// TwinCAT 3 PLC project Tc3_Logging
// Title: Tc3_Logging
// Company: www.peterzerlauth.com
// Author: Peter Zerlauth
// ProjectVersion: 0.0.0.8
// Description: Tc3_Logging – TwinCAT 3 Event Logging Framework Copyright (c) Peter Zerlauth This component is provided under a Dual Licensing Model: 1. GPLv3 Open-Source License - Free for personal, educational, and non-commercial use. - Commercial use allowed only if the entire application is published under GPLv3, including all modifications to this code. - Requires full disclosure of source code for derivative works. 2. Commercial License - Required for integration into proprietary or closed-source products. - Removes all GPLv3 copyleft obligations. - Includes optional warranty, professional support, and long-term maintenance options. For commercial licensing, contact: info@peterzerlauth.com By using this Function Block you agree to the terms of the selected license.
// ProgramVersion: 3.1.4026.24
// libraries:
//   SysDir, * (System)
//   SysFile, * (System)
//   Tc2_Standard, * (Beckhoff Automation GmbH)
//   Tc2_System, * (Beckhoff Automation GmbH)
//   Tc2_Utilities, * (Beckhoff Automation GmbH)
//   Tc3_EventLogger, * (Beckhoff Automation GmbH)
//   Tc3_Module, * (Beckhoff Automation GmbH)
// project tree:
//   Argument/ FB_Argument.TcPOU, I_Argument.TcIO
//   Event/ I_Event.TcIO (not stored), FB_Event.TcPOU (not stored)
//   Global Variables/ GVL.TcGVL
//   Helpers/File/ E_FileState.TcDUT, FB_File.TcPOU, I_File.TcIO
//   Helpers/ F_Filter.TcPOU, F_Hash.TcPOU, F_InstancePath.TcPOU, F_Log.TcPOU, F_Print.TcPOU, F_Remove.TcPOU, LogLevel_To_Severity.TcPOU
//   Logger/ E_LogLevel.TcDUT, I_Logger.TcIO
//   Logger/FileLogger/ FB_FileLogger.TcPOU
//   Logger/HmiLogger/ FB_HmiLogger.TcPOU
//   Logger/Manager/ FB_LoggerManager.TcPOU
//   Logger/TcLogger/ FB_TcLogger.TcPOU
//   Message/ FB_Message.TcPOU
//   Project Information/ F_GetCompany.TcPOU, F_GetTitle.TcPOU, F_GetVersion.TcPOU
//   Version/ Global_Version.TcGVL
// (motion and I/O tree: see PLC project plc01)
// real-time tasks:
//   TASK SlowTask: cycle T#20ms, priority 20, ADS port 350
//   TASK FastTask: cycle T#1ms, priority 1, ADS port 351

// ---- Helpers/File/E_FileState.TcDUT
{attribute 'qualified_only'}
{attribute 'strict'}
{attribute 'to_string'}
TYPE E_FileState :
(
    OK := 0,             // File could be opened
    NO_FILE := 1,        // No file available
    ILLEGAL_POS := 2,    // Illegal position in the file
    FULL := 3,           // No more space on the filesystem
    EOF := 4             // End of file reached
) UDINT;
END_TYPE

// ---- Logger/E_LogLevel.TcDUT
{attribute 'qualified_only'}
{attribute 'strict'}
{attribute 'to_string'}
TYPE E_LogLevel :
(
    Verbose 	:= 1,
    Info  		:= 2,
    Warning  	:= 3,
    Error 		:= 4,
    Critical 	:= 5
);
END_TYPE

// ---- Global Variables/GVL.TcGVL
{attribute 'no-analysis'}
{attribute 'qualified_only'} 
VAR_GLOBAL
	{attribute 'hide'} 
	aBuffer:				ARRAY[0..99] OF FB_Message;
	{attribute 'hide'} 
    nBuffer:				UINT := 0;
	{attribute 'hide'} 
	nTimestamp:				Tc2_Utilities.T_FILETIME64;	
	{attribute 'hide'} 
	nFunction:				Tc2_Utilities.T_FILETIME64;		
END_VAR

// ---- Version/Global_Version.TcGVL
{attribute 'TcGenerated'}
{attribute 'no-analysis'}
{attribute 'linkalways'}
// This function has been automatically generated from the project information.
VAR_GLOBAL CONSTANT
	{attribute 'const_non_replaced'}
	stLibVersion_Tc3_Logging : ST_LibVersion := (iMajor := 0, iMinor := 0, iBuild := 0, iRevision := 8, nFlags := 0, sVersion := '0.0.0.8');
END_VAR

// ---- Argument/I_Argument.TcIO
INTERFACE I_Argument

METHOD PUBLIC M_AddBOOL : I_Argument
VAR_INPUT
	bValue:				BOOL;
END_VAR
END_METHOD

METHOD PUBLIC M_AddINT : I_Argument
VAR_INPUT
	nValue:				LINT;
END_VAR
END_METHOD

METHOD PUBLIC M_AddREAL : I_Argument
VAR_INPUT
	fValue:				LREAL;
	nDecimals:			USINT;
END_VAR
END_METHOD

METHOD PUBLIC M_AddSTRING : I_Argument
VAR_INPUT
	sValue:				STRING(255);
END_VAR
END_METHOD

METHOD PUBLIC M_AddTIME : I_Argument
VAR_INPUT
	tValue:				TIME;
END_VAR
END_METHOD

METHOD PUBLIC M_Clear : I_Argument
VAR_INPUT
END_VAR
END_METHOD

PROPERTY PUBLIC P_Value : string(255)
GET
END_GET
END_PROPERTY

END_INTERFACE

// ---- Helpers/File/I_File.TcIO
INTERFACE I_File

// close file
METHOD PUBLIC M_Close : BOOL
VAR_INPUT
END_VAR
END_METHOD

// Delete file
METHOD PUBLIC M_Delete : BOOL
VAR_INPUT
    sFileName : STRING(255);
END_VAR
END_METHOD

// get file size
METHOD PUBLIC M_GetSize : UDINT
VAR_INPUT
END_VAR
END_METHOD

// Open file
METHOD PUBLIC M_Open : BOOL
VAR_INPUT
    sFileName:				STRING(255);
	eMode: 					SysFile.ACCESS_MODE := SysFile.AM_APPEND_PLUS;
END_VAR
END_METHOD

// Read file
METHOD PUBLIC M_Read : BOOL
VAR_INPUT
END_VAR
END_METHOD

// state of file
METHOD PUBLIC M_Status : E_FileState
VAR_INPUT
END_VAR
END_METHOD

// Write file
METHOD PUBLIC M_Write : BOOL
VAR_INPUT
	pBuffer:	POINTER TO BYTE;
    nSize:     	UDINT;
END_VAR
END_METHOD

END_INTERFACE

// ---- Logger/I_Logger.TcIO
INTERFACE I_Logger

METHOD PUBLIC M_Log : BOOL
VAR_INPUT
	fbMessage:			FB_Message;
END_VAR
END_METHOD

END_INTERFACE

// ---- Message/FB_Message.TcPOU
{attribute 'analysis' := '-33'}
// Payload for events
FUNCTION_BLOCK FB_Message
VAR_INPUT
	eLogLevel:			E_LogLevel;
	{attribute 'displaymode':='hex'}
	nID:				UDINT;
	nTimestamp:			Tc2_Utilities.T_FILETIME64;	
	sSource:			STRING(255);
	sType:				STRING(255);
	sMessage:			STRING(255);
	sDefault:			STRING(255);
	sArguments:			STRING(255);
	bActive:			BOOL;
END_VAR
VAR_OUTPUT
END_VAR
VAR
END_VAR
(*
    Tc3_Event – TwinCAT 3 Event Logging Framework
    Copyright (c) Peter Zerlauth

    This component is provided under a Dual Licensing Model:

    1. GPLv3 Open-Source License
       - Free for personal, educational, and non-commercial use.
       - Commercial use allowed only if the entire application is published
         under GPLv3, including all modifications to this code.
       - Requires full disclosure of source code for derivative works.

    2. Commercial License
       - Required for integration into proprietary or closed-source products.
       - Removes all GPLv3 copyleft obligations.
       - Includes optional warranty, professional support, and long-term
         maintenance options.

    For commercial licensing, contact:
        info@peterzerlauth.com

    By using this Function Block you agree to the terms of the selected license.
*)

END_FUNCTION_BLOCK

// ---- Argument/FB_Argument.TcPOU
{attribute 'no_explicit_call' := 'do not call this POU directly'}
// Store arguments in a single string seperated by $R
FUNCTION_BLOCK FB_Argument IMPLEMENTS I_Argument
VAR_INPUT
END_VAR
VAR_OUTPUT
END_VAR
VAR
	sValue:					STRING(255);		// storage for arguments
END_VAR
(*
    Tc3_Event – TwinCAT 3 Event Logging Framework
    Copyright (c) Peter Zerlauth

    This component is provided under a Dual Licensing Model:

    1. GPLv3 Open-Source License
       - Free for personal, educational, and non-commercial use.
       - Commercial use allowed only if the entire application is published
         under GPLv3, including all modifications to this code.
       - Requires full disclosure of source code for derivative works.

    2. Commercial License
       - Required for integration into proprietary or closed-source products.
       - Removes all GPLv3 copyleft obligations.
       - Includes optional warranty, professional support, and long-term
         maintenance options.

    For commercial licensing, contact:
        info@peterzerlauth.com

    By using this Function Block you agree to the terms of the selected license.
*)

// add boolean value to arguments
METHOD PUBLIC M_AddBOOL : I_Argument
VAR_INPUT
	bValue:				BOOL;		// Boolean input value
END_VAR
sValue:= CONCAT(sValue, BOOL_TO_STRING(bValue));			// convert
sValue:= CONCAT(sValue, '$R');								// add separator
M_AddBOOL:= THIS^;
END_METHOD

// add int value to arguments
METHOD PUBLIC M_AddINT : I_Argument
VAR_INPUT
	nValue:				LINT;		// Integer input value
END_VAR
VAR
	sTemp: 			STRING;
END_VAR
sValue:= CONCAT(sValue, CONCAT(LINT_TO_STRING(nValue), '$R'));	// add new arg
M_AddINT:= THIS^;
END_METHOD

// add real value to arguments
METHOD PUBLIC M_AddREAL : I_Argument
VAR_INPUT
	fValue:				LREAL;		// Real input value
	nDecimals:			USINT;		// Decimals afer .
END_VAR
VAR
	sTemp: 			STRING;
END_VAR
sValue:= CONCAT(sValue, CONCAT(LREAL_TO_FMTSTR(fValue, nDecimals, TRUE), '$R'));				// add new arg
M_AddREAL:= THIS^;
END_METHOD

// add string value to arguments
METHOD PUBLIC M_AddSTRING : I_Argument
VAR_INPUT
	sValue:				STRING(255);		// String input value
END_VAR
THIS^.sValue:= CONCAT(THIS^.sValue, CONCAT(sValue, '$R'));				// add separator 
M_AddSTRING:= THIS^;
END_METHOD

// add time value to arguments
METHOD PUBLIC M_AddTIME : I_Argument
VAR_INPUT
	tValue:				TIME;		// Time input value
END_VAR
sValue:= CONCAT(sValue, CONCAT(TIME_TO_STRING(tValue), '$R'));				// add separator
M_AddTIME:= THIS^;
END_METHOD

// Clear arguments
METHOD PUBLIC M_Clear : I_Argument
VAR_INPUT
END_VAR
sValue:= '';
M_Clear:= THIS^;
END_METHOD

// Returns the list with arguments
PROPERTY PUBLIC P_Value : STRING(255)
GET
P_Value:= sValue;
END_GET
END_PROPERTY

END_FUNCTION_BLOCK

// ---- Helpers/File/FB_File.TcPOU
// SysFile from codesys
{attribute 'no_explicit_call' := 'do not call this POU directly'} 
FUNCTION_BLOCK FB_File IMPLEMENTS I_File
VAR_INPUT
END_VAR
VAR_OUTPUT
    pBuffer:				POINTER TO BYTE;
    nBuffer:				UDINT;	
	bError:					BOOL;
END_VAR
VAR
	sFileName:				STRING(255);
	eMode: 					SysFile.ACCESS_MODE := SysFile.AM_APPEND_PLUS;
    hFile: 					SysFile.SysTypes.RTS_IEC_HANDLE;
	nResult:				SysFile.SysTypes.RTS_IEC_RESULT;
	{attribute 'hide'} 
	pResult:				POINTER TO SysFile.SysTypes.RTS_IEC_RESULT:= ADR(nResult);
END_VAR

// https://peterzerlauth.com/

//FB_Exit must be implemented explicitly. If there is an implementation, then the
//method is called before the controller removes the code of the function block instance
//(implicit call). The return value is not evaluated.
// Try to close and reset on exit
METHOD FB_Exit: BOOL
VAR_INPUT
    bInCopyCode: BOOL;  // TRUE: the exit method is called in order to leave the instance which will be copied afterwards (online change).  
END_VAR
M_Reset();
END_METHOD

// Closes the file if opened
METHOD PUBLIC M_Close : BOOL
VAR_INPUT
END_VAR
IF hFile > 0 THEN
   nResult:= SysFile.SysFileClose(hFile);
   IF nResult = 0 THEN
	   hFile:= 0;
	   M_Close:= TRUE;
   ELSE
	    bError := TRUE;
   END_IF
END_IF
END_METHOD

// Delete file
METHOD PUBLIC M_Delete : BOOL
VAR_INPUT
    sFileName : STRING(255);
END_VAR
IF hFile > 0 THEN
	M_Close();
END_IF

nResult:= SysFile.SysFileDelete(sFileName);
IF nResult = 0 THEN
	M_Delete:= TRUE;
ELSE
    bError := TRUE;
END_IF
END_METHOD

// Get file size
METHOD PUBLIC M_GetSize : UDINT
VAR_INPUT
END_VAR
M_GetSize:= LWORD_TO_UDINT(SysFile.SysFileGetSize(sFileName, pResult));

IF nResult <> 0 THEN
	bError := TRUE;
END_IF
END_METHOD

// Open file
METHOD PUBLIC M_Open : BOOL
VAR_INPUT
    sFileName:				STRING(255);					// file path
	eMode: 					SysFile.ACCESS_MODE := SysFile.AM_APPEND_PLUS;	// file mode
END_VAR
IF hFile = 0 THEN
	THIS^.eMode:= eMode;
	hFile := SysFile.SysFileOpen(sFileName, eMode, pResult);
	IF hFile = SysFile.SysTypes.RTS_INVALID_HANDLE  THEN
		bError := TRUE;
		RETURN;
	END_IF

   IF nResult = 0 THEN
	   THIS^.sFileName:= sFileName;
	   M_Open:= TRUE;
   ELSE
	    bError := TRUE;
   END_IF
ELSE 
	IF THIS^.sFileName = sFileName THEN
		M_Open:= TRUE;
	END_IF
END_IF
END_METHOD

// Read file
METHOD PUBLIC M_Read : BOOL
VAR_INPUT
END_VAR
IF pBuffer <> 0 THEN
	__DELETE(pBuffer);
	nBuffer:= 0;
END_IF

nBuffer:= M_GetSize();

IF nBuffer > 0 THEN
    pBuffer:= __NEW(BYTE, nBuffer);
	IF pBuffer = 0 THEN
		RETURN;
	END_IF
END_IF

IF M_Read = 0 THEN
	M_Read := TRUE;
ELSE
	bError:= TRUE;
END_IF
END_METHOD

// Reset all 
METHOD PUBLIC M_Reset : BOOL
VAR_INPUT
END_VAR
IF pBuffer <> 0 THEN
	__DELETE(pBuffer);
	nBuffer:= 0;
END_IF

M_Close();

bError:= FALSE;
M_Reset:= TRUE;
END_METHOD

// File status
METHOD PUBLIC M_Status : E_FileState
VAR_INPUT
END_VAR
VAR 
	nState:				SysFile.SYS_FILE_STATUS;
END_VAR
bError := FALSE;
nResult := 0; // This function does not use pResult

IF hFile < 0 THEN
   nState := SysFile.SysFileGetStatus(hFile);
   CASE nState OF
	   SysFile.SYS_FILE_STATUS.FS_OK:
   			M_Status:= E_FileState.OK;
			
	   SysFile.SYS_FILE_STATUS.FS_NO_FILE:
			M_Status:= E_FileState.NO_FILE;
			
	   SysFile.SYS_FILE_STATUS.FS_ILLEGAL_POS:
			M_Status:= E_FileState.ILLEGAL_POS;   
			
	   SysFile.SYS_FILE_STATUS.FS_FULL:
			M_Status:= E_FileState.FULL; 
			
	   SysFile.SYS_FILE_STATUS.FS_EOF:   
			M_Status:= E_FileState.EOF;
 
   END_CASE
   
END_IF
END_METHOD

// Writes content to a file
METHOD PUBLIC M_Write : BOOL
VAR_INPUT
	pBuffer:	POINTER TO BYTE;
    nSize:     	UDINT;
END_VAR
IF pBuffer = 0 OR nSize = 0 THEN
    RETURN;
END_IF

IF hFile > 0 THEN
	SysFile.SysFileWrite(hFile := hFile, pbyBuffer := pBuffer, ulSize := nSize, pResult := pResult);
END_IF

IF nResult = 0 THEN
	M_Write := TRUE;
ELSE
	bError:= TRUE;
END_IF
END_METHOD

END_FUNCTION_BLOCK

// ---- Helpers/F_Filter.TcPOU
// Filter messages, if already existing
FUNCTION F_Filter : BOOL
VAR_INPUT
	fbMessage:			FB_Message; // Input message
END_VAR
VAR
    nIndex:				UINT;	// Index counter
END_VAR
(*
    Tc3_Event – TwinCAT 3 Event Logging Framework
    Copyright (c) Peter Zerlauth

    This component is provided under a Dual Licensing Model:

    1. GPLv3 Open-Source License
       - Free for personal, educational, and non-commercial use.
       - Commercial use allowed only if the entire application is published
         under GPLv3, including all modifications to this code.
       - Requires full disclosure of source code for derivative works.

    2. Commercial License
       - Required for integration into proprietary or closed-source products.
       - Removes all GPLv3 copyleft obligations.
       - Includes optional warranty, professional support, and long-term
         maintenance options.

    For commercial licensing, contact:
        info@peterzerlauth.com

    By using this Function Block you agree to the terms of the selected license.
*)

nIndex := 0;
WHILE nIndex < GVL.nBuffer DO
	// check id first, more performance than a string comparison
    IF GVL.aBuffer[nIndex].nID = fbMessage.nID THEN
		IF GVL.aBuffer[nIndex].sSource = fbMessage.sSource THEN
			GVL.aBuffer[nIndex].bActive := TRUE;
			F_Filter := TRUE;
			RETURN;  // Message found
		END_IF
    END_IF
    nIndex := nIndex + 1;
END_WHILE

END_FUNCTION

// ---- Helpers/F_Hash.TcPOU
// Calculate hash value, same as the posershell sript
FUNCTION F_Hash : UDINT
VAR_INPUT
    sInput:					STRING(255);   				// input string to hash
END_VAR
VAR
    nPower:				ULINT := 37;
    nModulo:			ULINT := 1000000009;
    nHash:				ULINT := 0;
    nPow:				ULINT := 1;
    nValue:				USINT;
    nIndex:				INT;
    nLength:			INT;
END_VAR
(*
    Tc3_Event – TwinCAT 3 Event Logging Framework
    Copyright (c) Peter Zerlauth

    This component is provided under a Dual Licensing Model:

    1. GPLv3 Open-Source License
       - Free for personal, educational, and non-commercial use.
       - Commercial use allowed only if the entire application is published
         under GPLv3, including all modifications to this code.
       - Requires full disclosure of source code for derivative works.

    2. Commercial License
       - Required for integration into proprietary or closed-source products.
       - Removes all GPLv3 copyleft obligations.
       - Includes optional warranty, professional support, and long-term
         maintenance options.

    For commercial licensing, contact:
        info@peterzerlauth.com

    By using this Function Block you agree to the terms of the selected license.
*)

nLength:= Len(sInput);
FOR nIndex := 0 TO nLength DO
	nValue := sInput[nIndex];
    nHash := (nHash + (nValue * nPow MOD nModulo)) MOD nModulo;
    nPow := (nPow * nPower) MOD nModulo;
END_FOR

F_Hash:= Ulint_to_Udint(nHash);

END_FUNCTION

// ---- Helpers/F_InstancePath.TcPOU
// Filter instance path, to something useful
FUNCTION F_InstancePath : STRING(255)
VAR_INPUT
	sInstancePath:			STRING(255);
END_VAR
VAR
    nPosition     : INT;
END_VAR
(*
    Tc3_Event – TwinCAT 3 Event Logging Framework
    Copyright (c) Peter Zerlauth

    This component is provided under a Dual Licensing Model:

    1. GPLv3 Open-Source License
       - Free for personal, educational, and non-commercial use.
       - Commercial use allowed only if the entire application is published
         under GPLv3, including all modifications to this code.
       - Requires full disclosure of source code for derivative works.

    2. Commercial License
       - Required for integration into proprietary or closed-source products.
       - Removes all GPLv3 copyleft obligations.
       - Includes optional warranty, professional support, and long-term
         maintenance options.

    For commercial licensing, contact:
        info@peterzerlauth.com

    By using this Function Block you agree to the terms of the selected license.
*)

F_InstancePath:= RIGHT(sInstancePath, LEN(sInstancePath) - FIND(sInstancePath, '.'));
F_InstancePath:= RIGHT(F_InstancePath, LEN(F_InstancePath) - FIND(F_InstancePath, '.'));

FOR nPosition:= LEN(F_InstancePath) TO 1 BY -1 DO
    IF F_InstancePath[nPosition] = 46 THEN
		F_InstancePath := LEFT(F_InstancePath, nPosition);
		RETURN;
	END_IF
END_FOR

END_FUNCTION

// ---- Helpers/F_Log.TcPOU
// Standalone logger, if no logger is attached to FB_Event, nice for tessting
FUNCTION F_Log : BOOL
VAR_INPUT
	fbMessage:			REFERENCE TO FB_Message;
END_VAR
VAR
	sMessage:			STRING(255):= 'Logger = 0 | ';
    nIndex:				UINT;
END_VAR
(*
    Tc3_Event – TwinCAT 3 Event Logging Framework
    Copyright (c) Peter Zerlauth

    This component is provided under a Dual Licensing Model:

    1. GPLv3 Open-Source License
       - Free for personal, educational, and non-commercial use.
       - Commercial use allowed only if the entire application is published
         under GPLv3, including all modifications to this code.
       - Requires full disclosure of source code for derivative works.

    2. Commercial License
       - Required for integration into proprietary or closed-source products.
       - Removes all GPLv3 copyleft obligations.
       - Includes optional warranty, professional support, and long-term
         maintenance options.

    For commercial licensing, contact:
        info@peterzerlauth.com

    By using this Function Block you agree to the terms of the selected license.
*)

// --- Build log line
sMessage:= CONCAT('Logger null | ', fbMessage.sSource);
sMessage:= CONCAT(sMessage, ': ');
sMessage:= CONCAT(sMessage, fbMessage.sDefault);

// --- Keep active
IF F_Filter(fbMessage) THEN 
	RETURN;
END_IF

// --- Add to buffer ---
IF GVL.nBuffer < 99 THEN
    GVL.aBuffer[GVL.nBuffer]:= fbMessage;
    GVL.aBuffer[GVL.nBuffer].nTimestamp := GVL.nTimestamp;
    GVL.nBuffer := GVL.nBuffer + 1;
END_IF

// --- Log message ---
CASE fbMessage.eLogLevel OF
    E_LogLevel.Verbose, E_LogLevel.Info:
        ADSLOGSTR(ADSLOG_MSGTYPE_HINT, '%s', sMessage);
    E_LogLevel.Warning:
        ADSLOGSTR(ADSLOG_MSGTYPE_WARN, '%s', sMessage);
    E_LogLevel.Error, E_LogLevel.Critical:
        ADSLOGSTR(ADSLOG_MSGTYPE_ERROR, '%s', sMessage);
END_CASE

// --- Remove outdated messages
F_Remove();

F_Log := TRUE;

END_FUNCTION

// ---- Helpers/F_Remove.TcPOU
// Removes outdated messages from the buffer
FUNCTION F_Remove : BOOL
VAR_INPUT
END_VAR
VAR
    nIndex:					UDINT;
END_VAR
(*
    Tc3_Event – TwinCAT 3 Event Logging Framework
    Copyright (c) Peter Zerlauth

    This component is provided under a Dual Licensing Model:

    1. GPLv3 Open-Source License
       - Free for personal, educational, and non-commercial use.
       - Commercial use allowed only if the entire application is published
         under GPLv3, including all modifications to this code.
       - Requires full disclosure of source code for derivative works.

    2. Commercial License
       - Required for integration into proprietary or closed-source products.
       - Removes all GPLv3 copyleft obligations.
       - Includes optional warranty, professional support, and long-term
         maintenance options.

    For commercial licensing, contact:
        info@peterzerlauth.com

    By using this Function Block you agree to the terms of the selected license.
*)

// just once a cycle
IF GVL.nFunction <> GVL.nTimestamp THEN
	GVL.nFunction:= GVL.nTimestamp;
	// Remove outdated messages
	WHILE nIndex < GVL.nBuffer DO
		IF (GVL.nTimestamp - GVL.aBuffer[nIndex].nTimestamp) > 1_000_000_000 THEN // 1 s = 1e9 ns
			// Shift remaining messages down
			MEMMOVE(ADR(GVL.aBuffer[nIndex]), ADR(GVL.aBuffer[nIndex + 1]), SIZEOF(FB_Message) * (GVL.nBuffer - nIndex - 1));
			GVL.nBuffer := GVL.nBuffer - 1;
			F_Remove := TRUE;
		ELSE
			nIndex := nIndex + 1;
		END_IF
	END_WHILE
END_IF

END_FUNCTION

// ---- Helpers/F_Print.TcPOU
// Helper to generate a message with replaced arguments
FUNCTION F_Print : STRING(255)
VAR_INPUT
    sMessage:				STRING(255);
    sArguments:				STRING(255);	// Arguments are separated by $R 
END_VAR
VAR
    sArg:					STRING; 		// single argument
    nPosition:				INT;         	// Position of the $R delimiter
    nPlaceholder:			INT;         	// Position of the %s placeholder
END_VAR
(*
    Tc3_Event – TwinCAT 3 Event Logging Framework
    Copyright (c) Peter Zerlauth

    This component is provided under a Dual Licensing Model:

    1. GPLv3 Open-Source License
       - Free for personal, educational, and non-commercial use.
       - Commercial use allowed only if the entire application is published
         under GPLv3, including all modifications to this code.
       - Requires full disclosure of source code for derivative works.

    2. Commercial License
       - Required for integration into proprietary or closed-source products.
       - Removes all GPLv3 copyleft obligations.
       - Includes optional warranty, professional support, and long-term
         maintenance options.

    For commercial licensing, contact:
        info@peterzerlauth.com

    By using this Function Block you agree to the terms of the selected license.
*)

// replace placeholders with arguments
F_Print := sMessage;

IF sArguments = '' THEN
    RETURN;
END_IF

nPosition := FIND(sArguments, '$R');
WHILE nPosition > 0 DO
    
    sArg := LEFT(sArguments, nPosition - 1);
    
    nPlaceholder := FIND(F_Print, '%s');
    IF nPlaceholder > 0 THEN
        F_Print := REPLACE(F_Print, sArg, 2, nPlaceholder);
    ELSE
        RETURN;
    END_IF
	
    sArguments := DELETE(sArguments, nPosition, 1);
    nPosition := FIND(sArguments, '$R');
    
END_WHILE

END_FUNCTION

// ---- Helpers/LogLevel_To_Severity.TcPOU
// Converts internal loglevel to twincat severity
FUNCTION LogLevel_To_Severity : TcEventSeverity
VAR_INPUT
	eLogLevel:				E_LogLevel;
END_VAR
VAR
END_VAR
(*
    Tc3_Event – TwinCAT 3 Event Logging Framework
    Copyright (c) Peter Zerlauth

    This component is provided under a Dual Licensing Model:

    1. GPLv3 Open-Source License
       - Free for personal, educational, and non-commercial use.
       - Commercial use allowed only if the entire application is published
         under GPLv3, including all modifications to this code.
       - Requires full disclosure of source code for derivative works.

    2. Commercial License
       - Required for integration into proprietary or closed-source products.
       - Removes all GPLv3 copyleft obligations.
       - Includes optional warranty, professional support, and long-term
         maintenance options.

    For commercial licensing, contact:
        info@peterzerlauth.com

    By using this Function Block you agree to the terms of the selected license.
*)

CASE eLogLevel OF
	E_LogLevel.Verbose:
		LogLevel_To_Severity:= TcEventSeverity.Verbose;
		
	E_LogLevel.Info:
		LogLevel_To_Severity:= TcEventSeverity.Info;
		
	E_LogLevel.Warning:
		LogLevel_To_Severity:= TcEventSeverity.Warning;
		
	E_LogLevel.Error:
		LogLevel_To_Severity:= TcEventSeverity.Error;
		
	E_LogLevel.Critical:
		LogLevel_To_Severity:= TcEventSeverity.Critical;
		
END_CASE

END_FUNCTION

// ---- Logger/FileLogger/FB_FileLogger.TcPOU
// Provide logging 
FUNCTION_BLOCK FB_FileLogger IMPLEMENTS I_Logger
VAR_INPUT
	sPathName:				STRING(255):= 'C:\tempx\logger.txt';
END_VAR
VAR
    {attribute 'hide'} 
	eLogLevel:				E_LogLevel:= E_LogLevel.Verbose;
	fbFile:					FB_File;
	nTimestamp: 			Tc2_Utilities.T_FILETIME64;
	aBuffer:				ARRAY[0..99] OF FB_Message;
    nBuffer:				UINT := 0;                     // Message count
END_VAR
(*
    Tc3_Event – TwinCAT 3 Event Logging Framework
    Copyright (c) Peter Zerlauth

    This component is provided under a Dual Licensing Model:

    1. GPLv3 Open-Source License
       - Free for personal, educational, and non-commercial use.
       - Commercial use allowed only if the entire application is published
         under GPLv3, including all modifications to this code.
       - Requires full disclosure of source code for derivative works.

    2. Commercial License
       - Required for integration into proprietary or closed-source products.
       - Removes all GPLv3 copyleft obligations.
       - Includes optional warranty, professional support, and long-term
         maintenance options.

    For commercial licensing, contact:
        info@peterzerlauth.com

    By using this Function Block you agree to the terms of the selected license.
*)

// https://peterzerlauth.com/

METHOD PUBLIC M_Log : BOOL
VAR_INPUT
	fbMessage:			FB_Message;
END_VAR
VAR
	nIndex: 		UINT;
	sLogLine:		STRING(255);
	stTimestamp: Tc2_Utilities.TIMESTRUCT;
END_VAR
// Log Level
IF eLogLevel > fbMessage.eLogLevel THEN
	M_Log:= TRUE;
	RETURN;
END_IF

nTimestamp:= fbMessage.nTimestamp;

// Skip if message already in buffer
nIndex := 0;
WHILE nIndex < nBuffer DO
	// check id first, more performance than a string comparison
    IF aBuffer[nIndex].nID = fbMessage.nID THEN
		IF aBuffer[nIndex].sSource = fbMessage.sSource THEN
			aBuffer[nIndex].bActive := TRUE;
			RETURN;  // Message found
		END_IF
    END_IF
    nIndex := nIndex + 1;
END_WHILE


// Add new message
IF nBuffer < 99 THEN
    aBuffer[nBuffer] := fbMessage;
    nBuffer := nBuffer + 1;
END_IF

// Format log line
stTimestamp:= FILETIME64_TO_SYSTEMTIME(fbMessage.nTimestamp);

// Year
sLogLine := CONCAT('[', WORD_TO_DECSTR(stTimestamp.wYear, 4));
sLogLine := CONCAT(sLogLine, '-');
sLogLine := CONCAT(sLogLine, WORD_TO_DECSTR(stTimestamp.wMonth, 2));
sLogLine := CONCAT(sLogLine, '-');
sLogLine := CONCAT(sLogLine, WORD_TO_DECSTR(stTimestamp.wDay, 2));
sLogLine := CONCAT(sLogLine, 'T');

// Time
sLogLine := CONCAT(sLogLine, WORD_TO_DECSTR(stTimestamp.wHour, 2));
sLogLine := CONCAT(sLogLine, ':');
sLogLine := CONCAT(sLogLine, WORD_TO_DECSTR(stTimestamp.wMinute, 2));
sLogLine := CONCAT(sLogLine, ':');
sLogLine := CONCAT(sLogLine, WORD_TO_DECSTR(stTimestamp.wSecond, 2));
sLogLine := CONCAT(sLogLine, '.');
sLogLine := CONCAT(sLogLine, WORD_TO_DECSTR(stTimestamp.wMilliseconds, 3));


sLogLine := CONCAT(sLogLine, '] ');
sLogLine := CONCAT(sLogLine, TO_STRING(fbMessage.eLogLevel));
sLogLine := CONCAT(sLogLine, ' [');
sLogLine := CONCAT(sLogLine, UDINT_TO_STRING(fbMessage.nID));
sLogLine := CONCAT(sLogLine, '] ');
sLogLine := CONCAT(sLogLine, fbMessage.sDefault);
sLogLine := CONCAT(sLogLine, '$R$N');

// Write once per new message
fbFile.M_Open(sPathName);
fbFile.M_Write(ADR(sLogLine), INT_TO_UINT(LEN(sLogLine)));
fbFile.M_Close();

// Remove expired messages (>1 s old)
// just once a cycle
IF nTimestamp <> fbMessage.nTimestamp THEN
	nTimestamp:= fbMessage.nTimestamp;
	// Remove outdated messages
	WHILE nIndex < nBuffer DO
		IF (nTimestamp - aBuffer[nIndex].nTimestamp) > 1_000_000_000 THEN // 1 s = 1e9 ns
			// Shift remaining messages down
			MEMMOVE(ADR(aBuffer[nIndex]), ADR(aBuffer[nIndex + 1]), SIZEOF(FB_Message) * (nBuffer - nIndex - 1));
			nBuffer := nBuffer - 1;
		ELSE
			nIndex := nIndex + 1;
		END_IF
	END_WHILE
END_IF

M_Log := TRUE;
END_METHOD

METHOD PRIVATE M_Reset : BOOL
VAR_INPUT
END_VAR
M_Reset:= TRUE;
END_METHOD

{attribute 'OPC.UA.DA.Property' := '1'}
{attribute 'monitoring' := 'call'}
PROPERTY PUBLIC P_LogLevel : E_LogLevel
GET
P_LogLevel:= eLogLevel;
END_GET
SET
eLogLevel:= P_LogLevel;
END_SET
END_PROPERTY

END_FUNCTION_BLOCK

// ---- Logger/HmiLogger/FB_HmiLogger.TcPOU
// Provide logging 
FUNCTION_BLOCK FB_HmiLogger IMPLEMENTS I_Logger
VAR
    {attribute 'hide'} 
	eLogLevel:				E_LogLevel:= E_LogLevel.Verbose;
	{attribute 'OPC.UA.DA.Property' := '1'}
	aMessages:				ARRAY[0..99] OF FB_Message; 	// Message store
	{attribute 'OPC.UA.DA.Property' := '1'}
    nMessages:				UINT := 0;                     // Message count
	{attribute 'hide'} 
	nIndex: 				UINT;
	{attribute 'hide'} 
	nTimestamp:				LINT;
END_VAR
(*
    Tc3_Event – TwinCAT 3 Event Logging Framework
    Copyright (c) Peter Zerlauth

    This component is provided under a Dual Licensing Model:

    1. GPLv3 Open-Source License
       - Free for personal, educational, and non-commercial use.
       - Commercial use allowed only if the entire application is published
         under GPLv3, including all modifications to this code.
       - Requires full disclosure of source code for derivative works.

    2. Commercial License
       - Required for integration into proprietary or closed-source products.
       - Removes all GPLv3 copyleft obligations.
       - Includes optional warranty, professional support, and long-term
         maintenance options.

    For commercial licensing, contact:
        info@peterzerlauth.com

    By using this Function Block you agree to the terms of the selected license.
*)

// https://peterzerlauth.com/

IF nTimestamp < TwinCAT_SystemInfoVarList._TaskInfo[GETCURTASKINDEXEX()].DcTaskTime THEN // 1 second = 1e9 ns
	nTimestamp := TwinCAT_SystemInfoVarList._TaskInfo[GETCURTASKINDEXEX()].DcTaskTime + 1000000000;
	nIndex:= 0;
	WHILE nIndex < nMessages DO
		IF aMessages[nIndex].bActive THEN
			IF aMessages[nIndex].eLogLevel <= E_LogLevel.Warning THEN
				aMessages[nIndex].bActive:= FALSE;
			END_IF
			nIndex := nIndex + 1;
		ELSE
			MEMMOVE(ADR(aMessages[nIndex]), ADR(aMessages[nIndex + 1]), SIZEOF(FB_Message) * (nMessages - nIndex));
			nMessages := nMessages - 1;
		END_IF
	END_WHILE
END_IF

METHOD PUBLIC M_Log : BOOL
VAR_INPUT
	fbMessage:			FB_Message;
END_VAR
VAR
END_VAR
// 555652537:= F_Hash('###Reset###');
IF fbMessage.nID = 555652537 THEN
	// handle reset
	M_Log:= M_Reset();
	RETURN;
END_IF


IF eLogLevel > fbMessage.eLogLevel THEN
	M_Log:= TRUE;
	RETURN;
END_IF

IF nMessages > 99 THEN 
	RETURN;
END_IF

// Skip if same sMessage already exists
nIndex := 0;
WHILE nIndex < nMessages DO
    IF aMessages[nIndex].nID = fbMessage.nID THEN
		IF aMessages[nIndex].sSource = fbMessage.sSource THEN
			aMessages[nIndex].bActive:= TRUE;
			M_Log := TRUE;
			RETURN; // message already in buffer
		END_IF
    END_IF
    nIndex := nIndex + 1;
END_WHILE


aMessages[nMessages]:= fbMessage;;
nMessages := nMessages + 1;
M_Log := TRUE;
END_METHOD

METHOD PRIVATE M_Reset : BOOL
VAR_INPUT
END_VAR
nIndex := 0;
WHILE nIndex < nMessages DO
    IF aMessages[nIndex].bActive = TRUE THEN
		aMessages[nIndex].bActive:= FALSE;
    END_IF
    nIndex := nIndex + 1;
END_WHILE
M_Reset:= TRUE;
END_METHOD

{attribute 'OPC.UA.DA.Property' := '1'}
{attribute 'monitoring' := 'call'}
PROPERTY PUBLIC P_LogLevel : E_LogLevel
GET
P_LogLevel:= eLogLevel;
END_GET
SET
eLogLevel:= P_LogLevel;
END_SET
END_PROPERTY

END_FUNCTION_BLOCK

// ---- Logger/Manager/FB_LoggerManager.TcPOU
{attribute 'no_explicit_call' := 'do not call this POU directly'} 
// Provide the functionality to use more than one Logger target
FUNCTION_BLOCK FB_LoggerManager IMPLEMENTS I_Logger
VAR
    {attribute 'hide'} 
	nLength:		INT;
	pList: 			POINTER TO I_Logger;
	aList:			POINTER TO POINTER TO ARRAY [0..24] OF I_Logger:=ADR(pList);
END_VAR
(*
    Tc3_Event – TwinCAT 3 Event Logging Framework
    Copyright (c) Peter Zerlauth

    This component is provided under a Dual Licensing Model:

    1. GPLv3 Open-Source License
       - Free for personal, educational, and non-commercial use.
       - Commercial use allowed only if the entire application is published
         under GPLv3, including all modifications to this code.
       - Requires full disclosure of source code for derivative works.

    2. Commercial License
       - Required for integration into proprietary or closed-source products.
       - Removes all GPLv3 copyleft obligations.
       - Includes optional warranty, professional support, and long-term
         maintenance options.

    For commercial licensing, contact:
        info@peterzerlauth.com

    By using this Function Block you agree to the terms of the selected license.
*)

METHOD FB_exit : BOOL
VAR_INPUT
	bInCopyCode : BOOL; // if TRUE, the exit method is called for exiting an instance that is copied afterwards (online change).
END_VAR
M_Clear();
END_METHOD

METHOD PUBLIC M_Add : BOOL
VAR_INPUT
	iLogger: 	I_Logger;
END_VAR
VAR
	pOldList: 	POINTER TO I_Logger;
END_VAR
IF iLogger <> 0 THEN
	// First Item
	IF pList = 0 THEN
		nLength:= nLength + 1;
		pList:= __NEW(POINTER TO I_Logger, DINT_TO_UDINT(nLength));
	ELSE
		// Item already in List
		IF M_Find(iLogger) = -1 THEN
			// backup 
			pOldList:= pList;
			// new Length
			nLength:= nLength + 1;
			// new pointer
			pList:= __NEW(POINTER TO I_Logger, DINT_TO_UDINT(nLength));
			// restore
			Memcpy(pList, pOldList, SIZEOF(pList) * DINT_TO_UDINT(nLength -1));
			// delete old
			__DELETE(pOldList);
		ELSE
			M_Add:= FALSE;	
			RETURN;
		END_IF
	END_IF
	IF pList = 0 THEN
		RETURN;
	END_IF
	// add new Object
	pList[nLength-1]:= iLogger;
	M_Add:= TRUE;
ELSE
	M_Add:= FALSE;	
END_IF
END_METHOD

METHOD PUBLIC M_Clear : bool
IF pList <> 0 THEN
	nLength:= 0;
	__DELETE(pList);
END_IF
M_Clear:= TRUE;
END_METHOD

METHOD PUBLIC M_Find : DINT
VAR_INPUT
	iLogger: 	I_Logger;
END_VAR
VAR
	nIndex: 	UINT;
END_VAR
// Object already in List
M_Find := -1;
WHILE nIndex < nLength DO
    IF (pList[nIndex] = iLogger) THEN
        M_Find := nIndex;
        RETURN;
    END_IF
	nIndex := nIndex + 1;
END_WHILE
END_METHOD

METHOD PUBLIC M_Index : I_Logger
VAR_INPUT
	nIndex: 	DINT;
END_VAR
IF (nIndex < nLength) THEN
	M_Index := pList[nIndex];
END_IF
END_METHOD

METHOD PUBLIC M_Log : BOOL
VAR_INPUT
	fbMessage:			FB_Message;
END_VAR
VAR
	nIndex:		INT;
END_VAR
WHILE nIndex < nLength DO
    pList[nIndex].M_Log(fbMessage);
	nIndex := nIndex + 1;
END_WHILE
END_METHOD

METHOD PUBLIC M_Remove : BOOL
VAR_INPUT
	iLogger: 	I_Logger;
END_VAR
VAR
	pOldList:			POINTER TO I_Logger;
	nPosition: 			DINT;
END_VAR
IF iLogger <> 0 THEN
	// First Item
	IF nLength >= 0 THEN
		// Item already in List
		nPosition:= M_Find(iLogger);
		IF nPosition <> -1 THEN
			// backup 
			pOldList:= pList;
			// new Length
			nLength:= nLength -1;
			// new pointer
			pList:= __NEW(POINTER TO I_Logger ,DINT_TO_UDINT(nLength));
			// restore lower part
			Memcpy(pList, pOldList, SIZEOF(pList) * DINT_TO_UDINT(nPosition));
			//pList[nPosition]:= iObject;
			Memcpy(pList + (SIZEOF(pList) * nPosition),pOldList + (SIZEOF(pList)*(nPosition + 1)), SIZEOF(pList) * DINT_TO_UDINT(nLength - nPosition));
			// delete old
			__DELETE(pOldList);
		ELSE
			M_Remove:= FALSE;	
			RETURN;
		END_IF
	ELSE
		M_Remove:= FALSE;	
		RETURN;
	END_IF
	M_Remove:= TRUE;
ELSE
	M_Remove:= FALSE;	
END_IF
END_METHOD

METHOD public M_Reset : BOOL
VAR_INPUT
END_VAR
VAR
	nIndex: 				UINT;
	fbReset:				FB_Message;
END_VAR
fbReset.bActive:= TRUE;
fbReset.sMessage:= '###Reset###';
fbReset.eLogLevel:= E_LogLevel.Error;
fbReset.nID:= F_Hash(fbReset.sMessage);
fbReset.nTimestamp:= 0;
fbReset.sArguments:= '';
fbReset.sDefault:= '';
fbReset.sSource:= '';
fbReset.sType:= 'FB_LoggerManager';

nIndex := 0;
M_Reset:= TRUE;
WHILE nIndex < nLength DO
    IF pList[nIndex].M_Log(fbReset) THEN
		;
	ELSE
		M_Reset:= FALSE;
	END_IF
    nIndex := nIndex + 1;
END_WHILE
END_METHOD

{attribute 'OPC.UA.DA.Property' := '1'}
{attribute 'monitoring' := 'call'}
PROPERTY PUBLIC P_Length : DINT
GET
P_Length:= nLength;
END_GET
END_PROPERTY

END_FUNCTION_BLOCK

// ---- Logger/TcLogger/FB_TcLogger.TcPOU
FUNCTION_BLOCK FB_TcLogger IMPLEMENTS I_Logger
VAR_INPUT
END_VAR
VAR_OUTPUT
END_VAR
VAR
END_VAR

METHOD PUBLIC M_Log : BOOL
VAR_INPUT
	fbMessage	: FB_Message;
END_VAR
VAR
	sMessage:			STRING;
END_VAR
// --- Build log line
sMessage:= CONCAT(fbMessage.sSource, ': ');
sMessage:= CONCAT(sMessage, fbMessage.sDefault);

// --- Keep active
IF F_Filter(fbMessage) THEN 
	RETURN;
END_IF

// --- Add to buffer ---
IF GVL.nBuffer < 99 THEN
    GVL.aBuffer[GVL.nBuffer]:= fbMessage;
    GVL.aBuffer[GVL.nBuffer].nTimestamp := GVL.nTimestamp;
    GVL.nBuffer := GVL.nBuffer + 1;
END_IF

// --- Log message ---
CASE fbMessage.eLogLevel OF
    E_LogLevel.Verbose, E_LogLevel.Info:
        ADSLOGSTR(ADSLOG_MSGTYPE_HINT, '%s', sMessage);
    E_LogLevel.Warning:
        ADSLOGSTR(ADSLOG_MSGTYPE_WARN, '%s', sMessage);
    E_LogLevel.Error, E_LogLevel.Critical:
        ADSLOGSTR(ADSLOG_MSGTYPE_ERROR, '%s', sMessage);
END_CASE

// --- Remove outdated messages
F_Remove();

M_Log:= TRUE;
END_METHOD

END_FUNCTION_BLOCK

// ---- Project Information/F_GetCompany.TcPOU
// This function has been automatically generated from the project information.
{attribute 'signature_flag' := '1073741824'}
{attribute 'TcGenerated'}
{attribute 'no-analysis'}
FUNCTION F_GetCompany : WSTRING
VAR_INPUT
	
END_VAR

F_GetCompany := "www.peterzerlauth.com";

END_FUNCTION

// ---- Project Information/F_GetTitle.TcPOU
// This function has been automatically generated from the project information.
{attribute 'signature_flag' := '1073741824'}
{attribute 'TcGenerated'}
{attribute 'no-analysis'}
FUNCTION F_GetTitle : WSTRING
VAR_INPUT
	
END_VAR

F_GetTitle := "Tc3_Logging";

END_FUNCTION

// ---- Project Information/F_GetVersion.TcPOU
// This function has been automatically generated from the project information.
{attribute 'signature_flag' := '1073741824'}
{attribute 'TcGenerated'}
{attribute 'no-analysis'}
FUNCTION F_GetVersion : ST_LibVersion
VAR_INPUT
	
END_VAR

F_GetVersion.iMajor := 0;
F_GetVersion.iMinor := 0;
F_GetVersion.iBuild := 0;
F_GetVersion.iRevision := 8;
F_GetVersion.sVersion := '0.0.0.8';
F_GetVersion.nFlags := 0;

END_FUNCTION
